SYSTEM FillingModule (* Module Filling, generated from its module specification *)
  (* Standard: 61499-2 *)
  APPLICATION Filling (* Module Filling on target pc (localhost, IO modbus; generated by modgen) *)
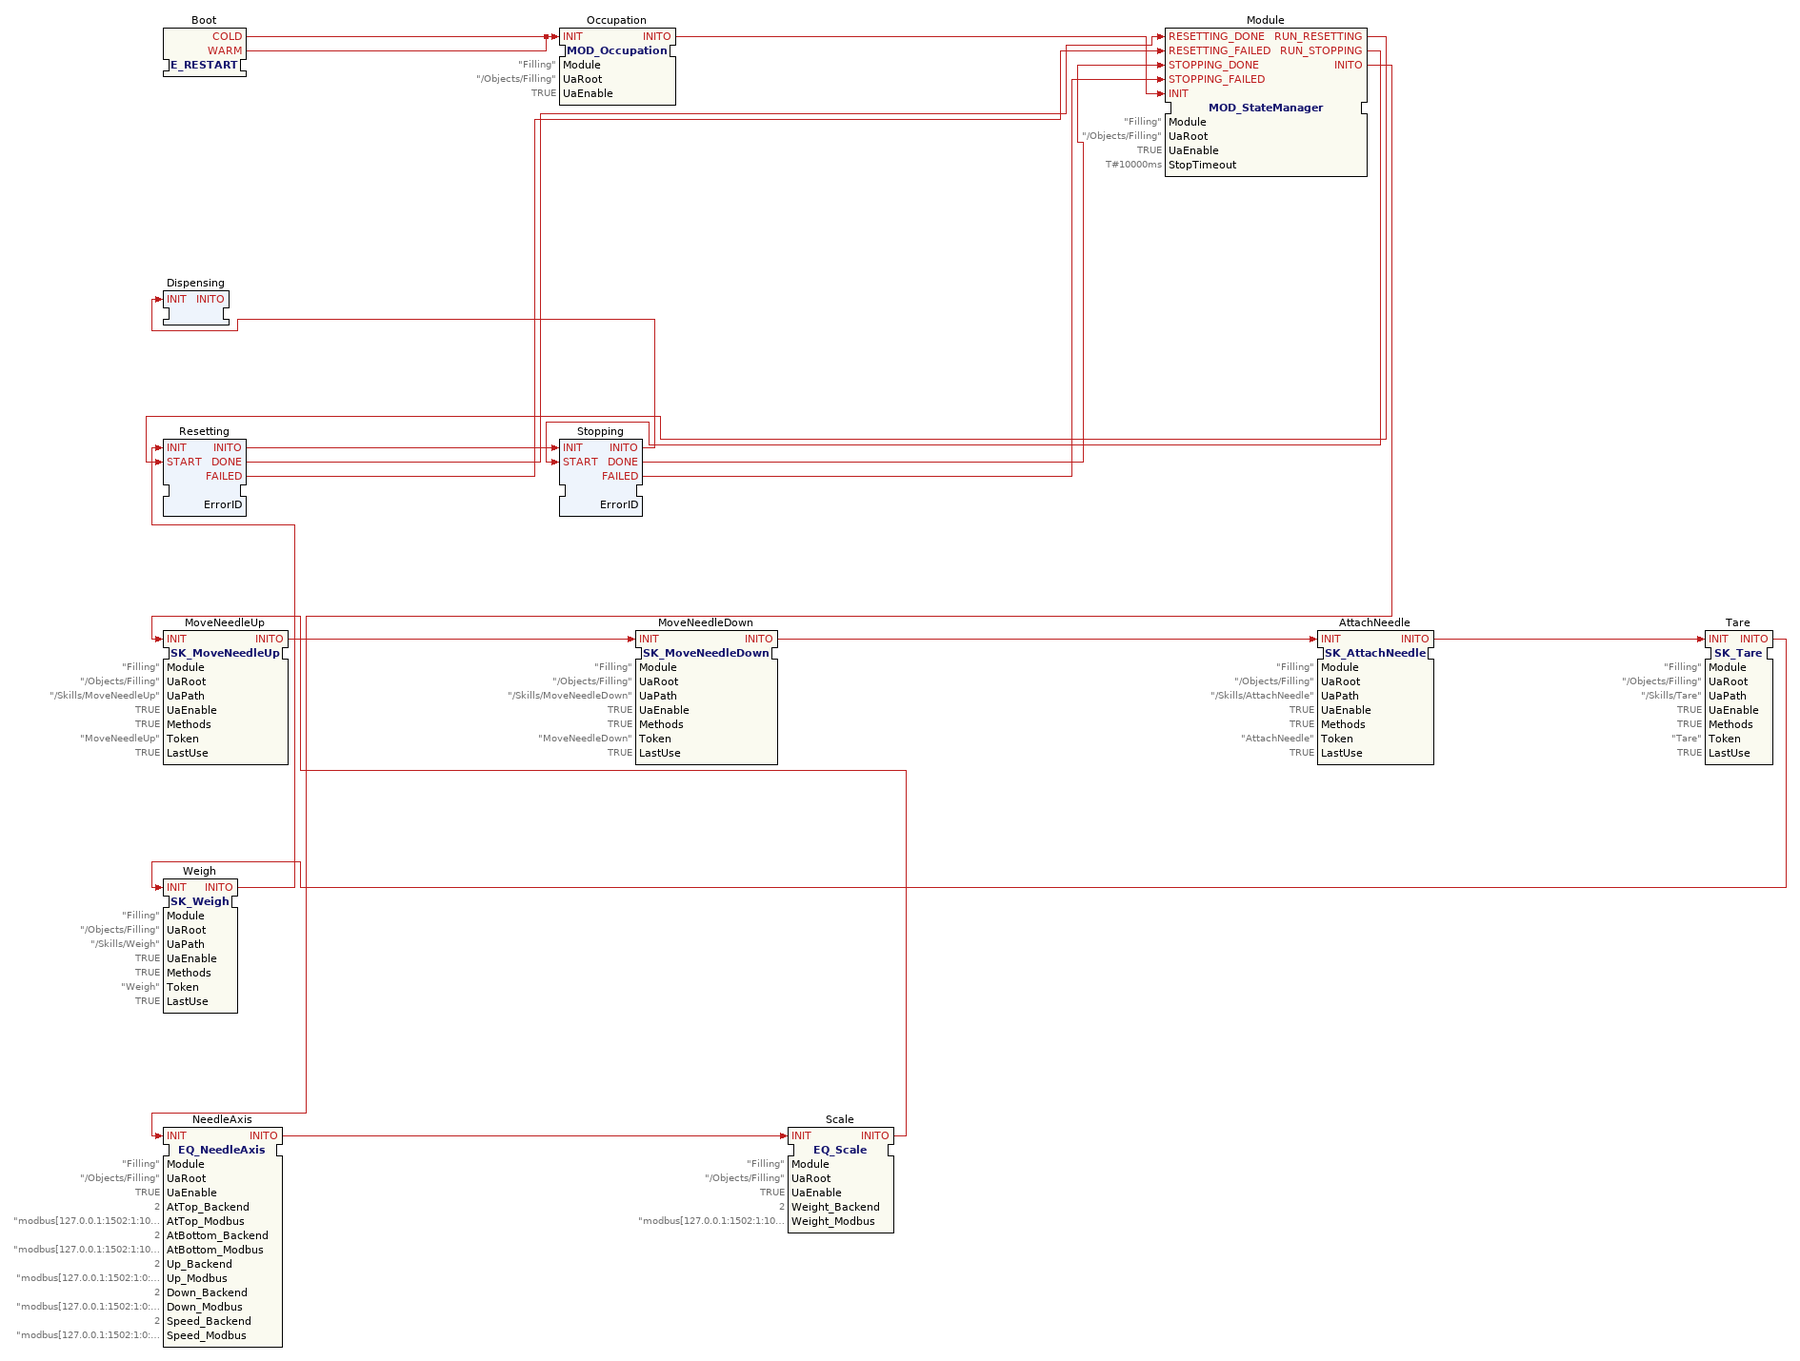
    (* Group ModuleLevel: Module level: occupation, PackML state manager, start-up and the target's IO lines *)
    (* Group ModuleLevelSkills: Module level skills: Control, Sequences (Execute, Stop) of skill primitives and Release; OPC UA /Skills/<name> *)
    (* Group Procedures: Procedures the module state manager runs while Resetting and Stopping *)
    (* Group SkillPrimitives: Skill primitives: one equipment command until a sensor or a time; OPC UA /Skills/<name> *)
    (* Group EquipmentIO: Equipment IO: the only owners of the IO points; skills send them output values over local channels *)
    FBS
      Boot : iec61499::events::E_RESTART; {SET_ATTRIBUTE(GroupName, ModuleLevel)}
      Occupation : modlib::MOD_Occupation(Module := "Filling", UaRoot := "/Objects/Filling", UaEnable := TRUE); {SET_ATTRIBUTE(GroupName, ModuleLevel)}
      Module : modlib::MOD_StateManager(Module := "Filling", UaRoot := "/Objects/Filling", UaEnable := TRUE, StopTimeout := T#10000ms); {SET_ATTRIBUTE(GroupName, ModuleLevel)}
      NeedleAxis : filling::EQ_NeedleAxis(Module := "Filling", UaRoot := "/Objects/Filling", UaEnable := TRUE, AtTop_Backend := 2, AtTop_Modbus := "modbus[127.0.0.1:1502:1:10:d0:]", AtBottom_Backend := 2, AtBottom_Modbus := "modbus[127.0.0.1:1502:1:10:d1:]", Up_Backend := 2, Up_Modbus := "modbus[127.0.0.1:1502:1:0::c0]", Down_Backend := 2, Down_Modbus := "modbus[127.0.0.1:1502:1:0::c1]", Speed_Backend := 2, Speed_Modbus := "modbus[127.0.0.1:1502:1:0::h0]"); {SET_ATTRIBUTE(GroupName, EquipmentIO)}
      Scale : filling::EQ_Scale(Module := "Filling", UaRoot := "/Objects/Filling", UaEnable := TRUE, Weight_Backend := 2, Weight_Modbus := "modbus[127.0.0.1:1502:1:10:i0:]"); {SET_ATTRIBUTE(GroupName, EquipmentIO)}
      MoveNeedleUp : filling::SK_MoveNeedleUp(Module := "Filling", UaRoot := "/Objects/Filling", UaPath := "/Skills/MoveNeedleUp", UaEnable := TRUE, Methods := TRUE, Token := "MoveNeedleUp", LastUse := TRUE); {SET_ATTRIBUTE(GroupName, SkillPrimitives)}
      MoveNeedleDown : filling::SK_MoveNeedleDown(Module := "Filling", UaRoot := "/Objects/Filling", UaPath := "/Skills/MoveNeedleDown", UaEnable := TRUE, Methods := TRUE, Token := "MoveNeedleDown", LastUse := TRUE); {SET_ATTRIBUTE(GroupName, SkillPrimitives)}
      AttachNeedle : filling::SK_AttachNeedle(Module := "Filling", UaRoot := "/Objects/Filling", UaPath := "/Skills/AttachNeedle", UaEnable := TRUE, Methods := TRUE, Token := "AttachNeedle", LastUse := TRUE); {SET_ATTRIBUTE(GroupName, SkillPrimitives)}
      Tare : filling::SK_Tare(Module := "Filling", UaRoot := "/Objects/Filling", UaPath := "/Skills/Tare", UaEnable := TRUE, Methods := TRUE, Token := "Tare", LastUse := TRUE); {SET_ATTRIBUTE(GroupName, SkillPrimitives)}
      Weigh : filling::SK_Weigh(Module := "Filling", UaRoot := "/Objects/Filling", UaPath := "/Skills/Weigh", UaEnable := TRUE, Methods := TRUE, Token := "Weigh", LastUse := TRUE); {SET_ATTRIBUTE(GroupName, SkillPrimitives)}
    END_FBS
    SUBAPPLICATION Resetting (* Procedure the module runs while Resetting *)
      {SET_ATTRIBUTE(GroupName, Procedures)}
      EVENT_INPUT
        INIT : EInit;
        START;
      END_EVENT
      EVENT_OUTPUT
        INITO : EInit;
        DONE;
        FAILED;
      END_EVENT
      VAR_OUTPUT
        ErrorID : UINT;
      END_VAR
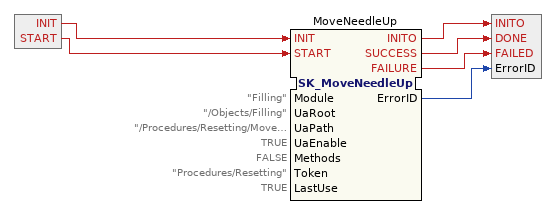
      FBS
        MoveNeedleUp : filling::SK_MoveNeedleUp(Module := "Filling", UaRoot := "/Objects/Filling", UaPath := "/Procedures/Resetting/MoveNeedleUp", UaEnable := TRUE, Methods := FALSE, Token := "Procedures/Resetting", LastUse := TRUE);
      END_FBS
      EVENT_CONNECTIONS
        INIT TO MoveNeedleUp.INIT;
        MoveNeedleUp.INITO TO INITO;
        START TO MoveNeedleUp.START;
        MoveNeedleUp.SUCCESS TO DONE;
        MoveNeedleUp.FAILURE TO FAILED;
      END_CONNECTIONS
      DATA_CONNECTIONS
        MoveNeedleUp.ErrorID TO ErrorID;
      END_CONNECTIONS
    END_SUBAPPLICATION
    SUBAPPLICATION Stopping (* Procedure the module runs while Stopping *)
      {SET_ATTRIBUTE(GroupName, Procedures)}
      EVENT_INPUT
        INIT : EInit;
        START;
      END_EVENT
      EVENT_OUTPUT
        INITO : EInit;
        DONE;
        FAILED;
      END_EVENT
      VAR_OUTPUT
        ErrorID : UINT;
      END_VAR
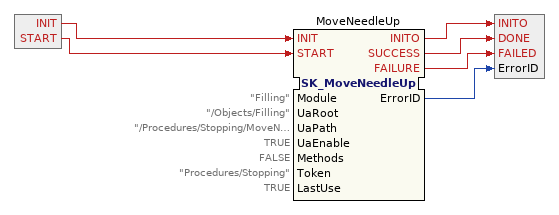
      FBS
        MoveNeedleUp : filling::SK_MoveNeedleUp(Module := "Filling", UaRoot := "/Objects/Filling", UaPath := "/Procedures/Stopping/MoveNeedleUp", UaEnable := TRUE, Methods := FALSE, Token := "Procedures/Stopping", LastUse := TRUE);
      END_FBS
      EVENT_CONNECTIONS
        INIT TO MoveNeedleUp.INIT;
        MoveNeedleUp.INITO TO INITO;
        START TO MoveNeedleUp.START;
        MoveNeedleUp.SUCCESS TO DONE;
        MoveNeedleUp.FAILURE TO FAILED;
      END_CONNECTIONS
      DATA_CONNECTIONS
        MoveNeedleUp.ErrorID TO ErrorID;
      END_CONNECTIONS
    END_SUBAPPLICATION
    SUBAPPLICATION Dispensing (* Module level skill Dispensing: Needle down, dispense the volume, needle up, weigh (runFillingCycle) *)
      {SET_ATTRIBUTE(GroupName, ModuleLevelSkills)}
      EVENT_INPUT
        INIT : EInit;
      END_EVENT
      EVENT_OUTPUT
        INITO : EInit;
      END_EVENT
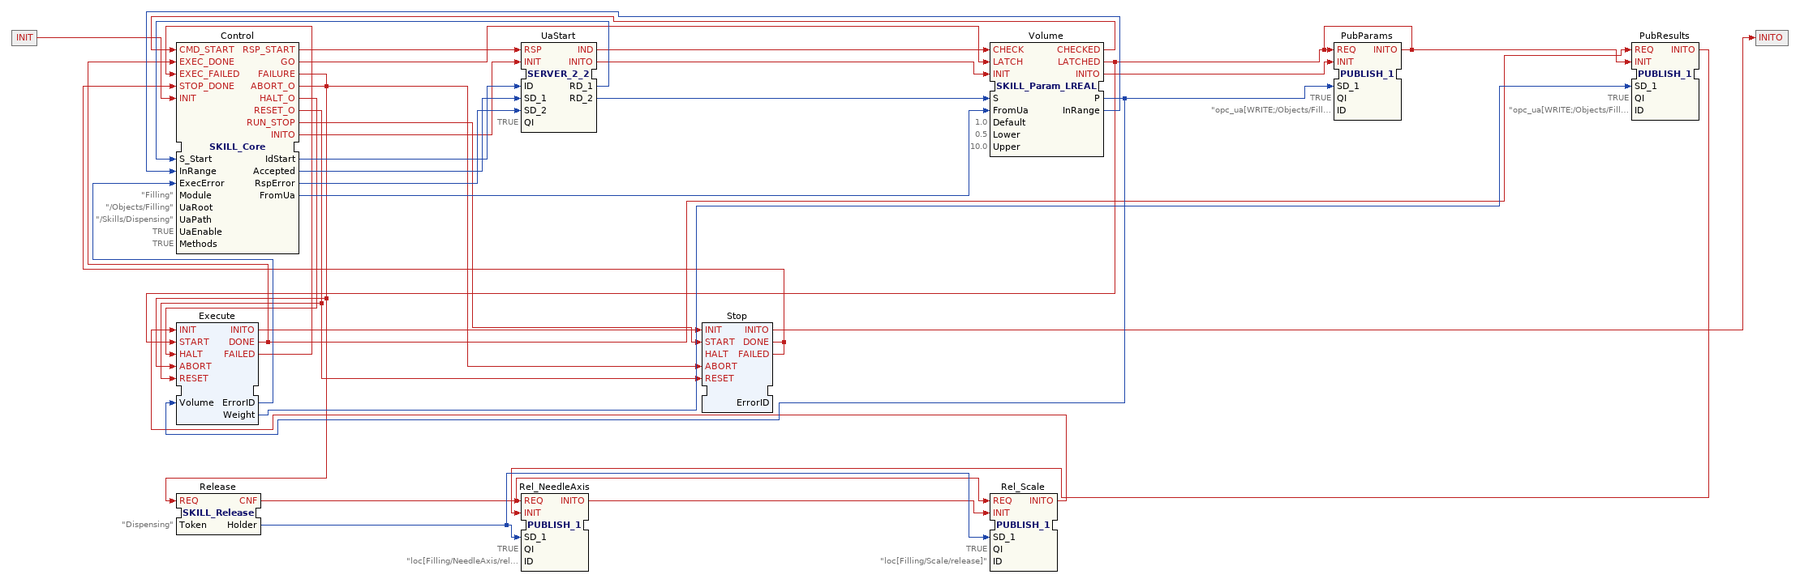
      (* Group SkillControl: State machine and OPC UA: Start(Session, parameters) with one block per parameter (range check, value for this run), Stop, Abort, Reset; State, parameters and results published *)
      (* Group Sequences: What the skill does: Execute, and Stop when it is interrupted; private skill primitives in order *)
      (* Group Releasing: After a failure or an abort: gives up the equipment the skill holds (all off, free again) *)
      FBS
        Control : modlib::SKILL_Core(Module := "Filling", UaRoot := "/Objects/Filling", UaPath := "/Skills/Dispensing", UaEnable := TRUE, Methods := TRUE); {SET_ATTRIBUTE(GroupName, SkillControl)}
        UaStart : iec61499::net::SERVER_2_2(QI := TRUE); {SET_ATTRIBUTE(GroupName, SkillControl)}
        Volume : modlib::SKILL_Param_LREAL(Default := 1.0, Lower := 0.5, Upper := 10.0); {SET_ATTRIBUTE(GroupName, SkillControl)}
        PubParams : iec61499::net::PUBLISH_1(QI := TRUE, ID := "opc_ua[WRITE;/Objects/Filling/Skills/Dispensing/Parameters/Volume]"); {SET_ATTRIBUTE(GroupName, SkillControl)}
        PubResults : iec61499::net::PUBLISH_1(QI := TRUE, ID := "opc_ua[WRITE;/Objects/Filling/Skills/Dispensing/Results/Weight]"); {SET_ATTRIBUTE(GroupName, SkillControl)}
        Release : modlib::SKILL_Release(Token := "Dispensing"); {SET_ATTRIBUTE(GroupName, Releasing)}
        Rel_NeedleAxis : iec61499::net::PUBLISH_1(QI := TRUE, ID := "loc[Filling/NeedleAxis/release]"); {SET_ATTRIBUTE(GroupName, Releasing)}
        Rel_Scale : iec61499::net::PUBLISH_1(QI := TRUE, ID := "loc[Filling/Scale/release]"); {SET_ATTRIBUTE(GroupName, Releasing)}
      END_FBS
      SUBAPPLICATION Execute (* Dispensing: execute sequence *)
        {SET_ATTRIBUTE(GroupName, Sequences)}
        EVENT_INPUT
          INIT : EInit;
          START;
          HALT;
          ABORT;
          RESET;
        END_EVENT
        EVENT_OUTPUT
          INITO : EInit;
          DONE;
          FAILED;
        END_EVENT
        VAR_INPUT
          Volume : LREAL;
        END_VAR
        VAR_OUTPUT
          ErrorID : UINT;
          Weight : LREAL;
        END_VAR
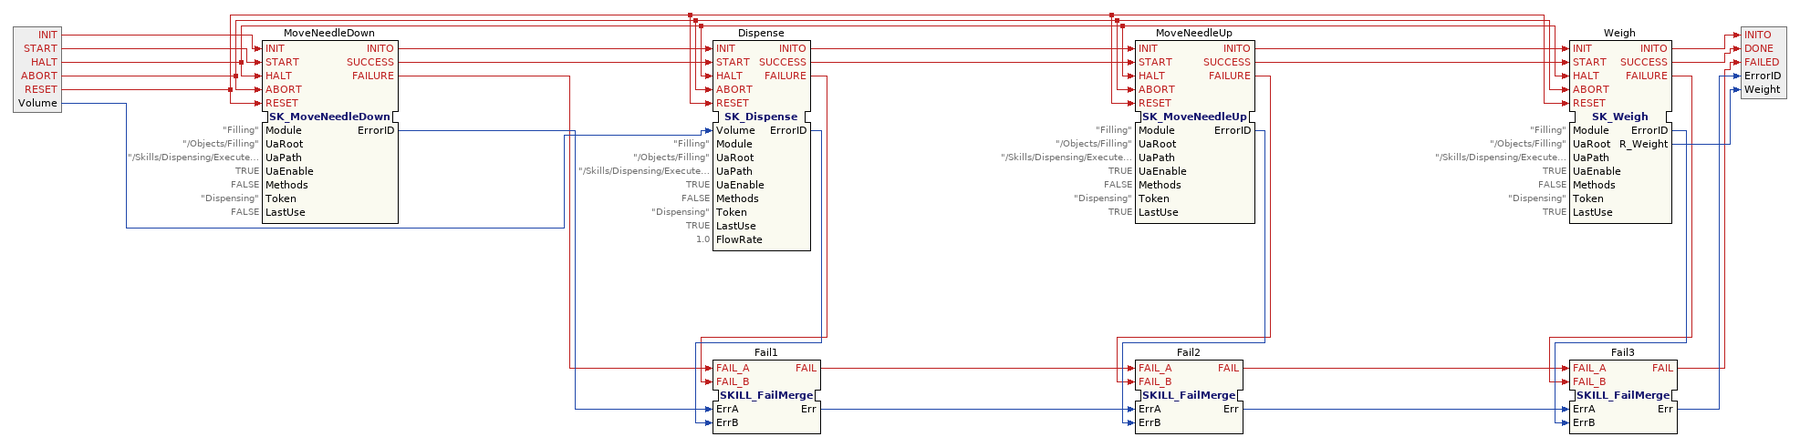
        FBS
          MoveNeedleDown : filling::SK_MoveNeedleDown(Module := "Filling", UaRoot := "/Objects/Filling", UaPath := "/Skills/Dispensing/Execute/MoveNeedleDown", UaEnable := TRUE, Methods := FALSE, Token := "Dispensing", LastUse := FALSE);
          Dispense : filling::SK_Dispense(Module := "Filling", UaRoot := "/Objects/Filling", UaPath := "/Skills/Dispensing/Execute/Dispense", UaEnable := TRUE, Methods := FALSE, Token := "Dispensing", LastUse := TRUE, FlowRate := 1.0);
          MoveNeedleUp : filling::SK_MoveNeedleUp(Module := "Filling", UaRoot := "/Objects/Filling", UaPath := "/Skills/Dispensing/Execute/MoveNeedleUp", UaEnable := TRUE, Methods := FALSE, Token := "Dispensing", LastUse := TRUE);
          Weigh : filling::SK_Weigh(Module := "Filling", UaRoot := "/Objects/Filling", UaPath := "/Skills/Dispensing/Execute/Weigh", UaEnable := TRUE, Methods := FALSE, Token := "Dispensing", LastUse := TRUE);
          Fail1 : modlib::SKILL_FailMerge;
          Fail2 : modlib::SKILL_FailMerge;
          Fail3 : modlib::SKILL_FailMerge;
        END_FBS
        EVENT_CONNECTIONS
          INIT TO MoveNeedleDown.INIT;
          Weigh.INITO TO INITO;
          START TO MoveNeedleDown.START;
          Weigh.SUCCESS TO DONE;
          MoveNeedleDown.INITO TO Dispense.INIT;
          MoveNeedleDown.SUCCESS TO Dispense.START;
          Dispense.INITO TO MoveNeedleUp.INIT;
          Dispense.SUCCESS TO MoveNeedleUp.START;
          MoveNeedleUp.INITO TO Weigh.INIT;
          MoveNeedleUp.SUCCESS TO Weigh.START;
          HALT TO MoveNeedleDown.HALT;
          HALT TO Dispense.HALT;
          HALT TO MoveNeedleUp.HALT;
          HALT TO Weigh.HALT;
          ABORT TO MoveNeedleDown.ABORT;
          ABORT TO Dispense.ABORT;
          ABORT TO MoveNeedleUp.ABORT;
          ABORT TO Weigh.ABORT;
          RESET TO MoveNeedleDown.RESET;
          RESET TO Dispense.RESET;
          RESET TO MoveNeedleUp.RESET;
          RESET TO Weigh.RESET;
          MoveNeedleDown.FAILURE TO Fail1.FAIL_A;
          Dispense.FAILURE TO Fail1.FAIL_B;
          Fail1.FAIL TO Fail2.FAIL_A;
          MoveNeedleUp.FAILURE TO Fail2.FAIL_B;
          Fail2.FAIL TO Fail3.FAIL_A;
          Weigh.FAILURE TO Fail3.FAIL_B;
          Fail3.FAIL TO FAILED;
        END_CONNECTIONS
        DATA_CONNECTIONS
          MoveNeedleDown.ErrorID TO Fail1.ErrA;
          Dispense.ErrorID TO Fail1.ErrB;
          Fail1.Err TO Fail2.ErrA;
          MoveNeedleUp.ErrorID TO Fail2.ErrB;
          Fail2.Err TO Fail3.ErrA;
          Weigh.ErrorID TO Fail3.ErrB;
          Fail3.Err TO ErrorID;
          Volume TO Dispense.Volume;
          Weigh.R_Weight TO Weight;
        END_CONNECTIONS
      END_SUBAPPLICATION
      SUBAPPLICATION Stop (* Dispensing: stop sequence *)
        {SET_ATTRIBUTE(GroupName, Sequences)}
        EVENT_INPUT
          INIT : EInit;
          START;
          HALT;
          ABORT;
          RESET;
        END_EVENT
        EVENT_OUTPUT
          INITO : EInit;
          DONE;
          FAILED;
        END_EVENT
        VAR_OUTPUT
          ErrorID : UINT;
        END_VAR
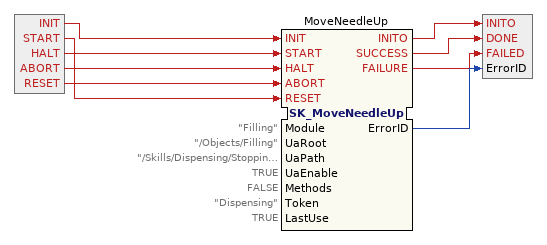
        FBS
          MoveNeedleUp : filling::SK_MoveNeedleUp(Module := "Filling", UaRoot := "/Objects/Filling", UaPath := "/Skills/Dispensing/Stopping/MoveNeedleUp", UaEnable := TRUE, Methods := FALSE, Token := "Dispensing", LastUse := TRUE);
        END_FBS
        EVENT_CONNECTIONS
          INIT TO MoveNeedleUp.INIT;
          MoveNeedleUp.INITO TO INITO;
          START TO MoveNeedleUp.START;
          MoveNeedleUp.SUCCESS TO DONE;
          HALT TO MoveNeedleUp.HALT;
          ABORT TO MoveNeedleUp.ABORT;
          RESET TO MoveNeedleUp.RESET;
          MoveNeedleUp.FAILURE TO FAILED;
        END_CONNECTIONS
        DATA_CONNECTIONS
          MoveNeedleUp.ErrorID TO ErrorID;
        END_CONNECTIONS
      END_SUBAPPLICATION
      EVENT_CONNECTIONS
        Control.RSP_START TO UaStart.RSP;
        UaStart.IND TO Volume.CHECK;
        Control.GO TO Volume.LATCH;
        Volume.CHECKED TO Control.CMD_START;
        Volume.LATCHED TO PubParams.REQ;
        PubParams.INITO TO PubParams.REQ;
        Execute.DONE TO PubResults.REQ;
        Control.FAILURE TO Release.REQ;
        Control.ABORT_O TO Release.REQ;
        Release.CNF TO Rel_NeedleAxis.REQ;
        Release.CNF TO Rel_Scale.REQ;
        Volume.LATCHED TO Execute.START;
        Control.HALT_O TO Execute.HALT;
        Control.ABORT_O TO Execute.ABORT;
        Control.RESET_O TO Execute.RESET;
        Execute.DONE TO Control.EXEC_DONE;
        Execute.FAILED TO Control.EXEC_FAILED;
        Control.RUN_STOP TO Stop.START;
        Control.ABORT_O TO Stop.ABORT;
        Control.RESET_O TO Stop.RESET;
        Stop.DONE TO Control.STOP_DONE;
        Stop.FAILED TO Control.STOP_DONE;
        INIT TO Control.INIT;
        Control.INITO TO UaStart.INIT;
        UaStart.INITO TO Volume.INIT;
        Volume.INITO TO PubParams.INIT;
        PubParams.INITO TO PubResults.INIT;
        PubResults.INITO TO Rel_NeedleAxis.INIT;
        Rel_NeedleAxis.INITO TO Rel_Scale.INIT;
        Rel_Scale.INITO TO Execute.INIT;
        Execute.INITO TO Stop.INIT;
        Stop.INITO TO INITO;
      END_CONNECTIONS
      DATA_CONNECTIONS
        Control.IdStart TO UaStart.ID;
        UaStart.RD_1 TO Control.S_Start;
        Control.Accepted TO UaStart.SD_1;
        Control.RspError TO UaStart.SD_2;
        UaStart.RD_2 TO Volume.S;
        Control.FromUa TO Volume.FromUa;
        Volume.P TO PubParams.SD_1;
        Volume.InRange TO Control.InRange;
        Execute.Weight TO PubResults.SD_1;
        Release.Holder TO Rel_NeedleAxis.SD_1;
        Release.Holder TO Rel_Scale.SD_1;
        Volume.P TO Execute.Volume;
        Execute.ErrorID TO Control.ExecError;
      END_CONNECTIONS
    END_SUBAPPLICATION
    EVENT_CONNECTIONS
      Boot.COLD TO Occupation.INIT;
      Boot.WARM TO Occupation.INIT;
      Module.RUN_RESETTING TO Resetting.START;
      Resetting.DONE TO Module.RESETTING_DONE;
      Resetting.FAILED TO Module.RESETTING_FAILED;
      Module.RUN_STOPPING TO Stopping.START;
      Stopping.DONE TO Module.STOPPING_DONE;
      Stopping.FAILED TO Module.STOPPING_FAILED;
      Occupation.INITO TO Module.INIT;
      Module.INITO TO NeedleAxis.INIT;
      NeedleAxis.INITO TO Scale.INIT;
      Scale.INITO TO MoveNeedleUp.INIT;
      MoveNeedleUp.INITO TO MoveNeedleDown.INIT;
      MoveNeedleDown.INITO TO AttachNeedle.INIT;
      AttachNeedle.INITO TO Tare.INIT;
      Tare.INITO TO Weigh.INIT;
      Weigh.INITO TO Resetting.INIT;
      Resetting.INITO TO Stopping.INIT;
      Stopping.INITO TO Dispensing.INIT;
    END_CONNECTIONS
  END_APPLICATION
  APPLICATION Filling_pi (* Module Filling on target pi (192.168.0.191, IO gpio; generated by modgen) *)
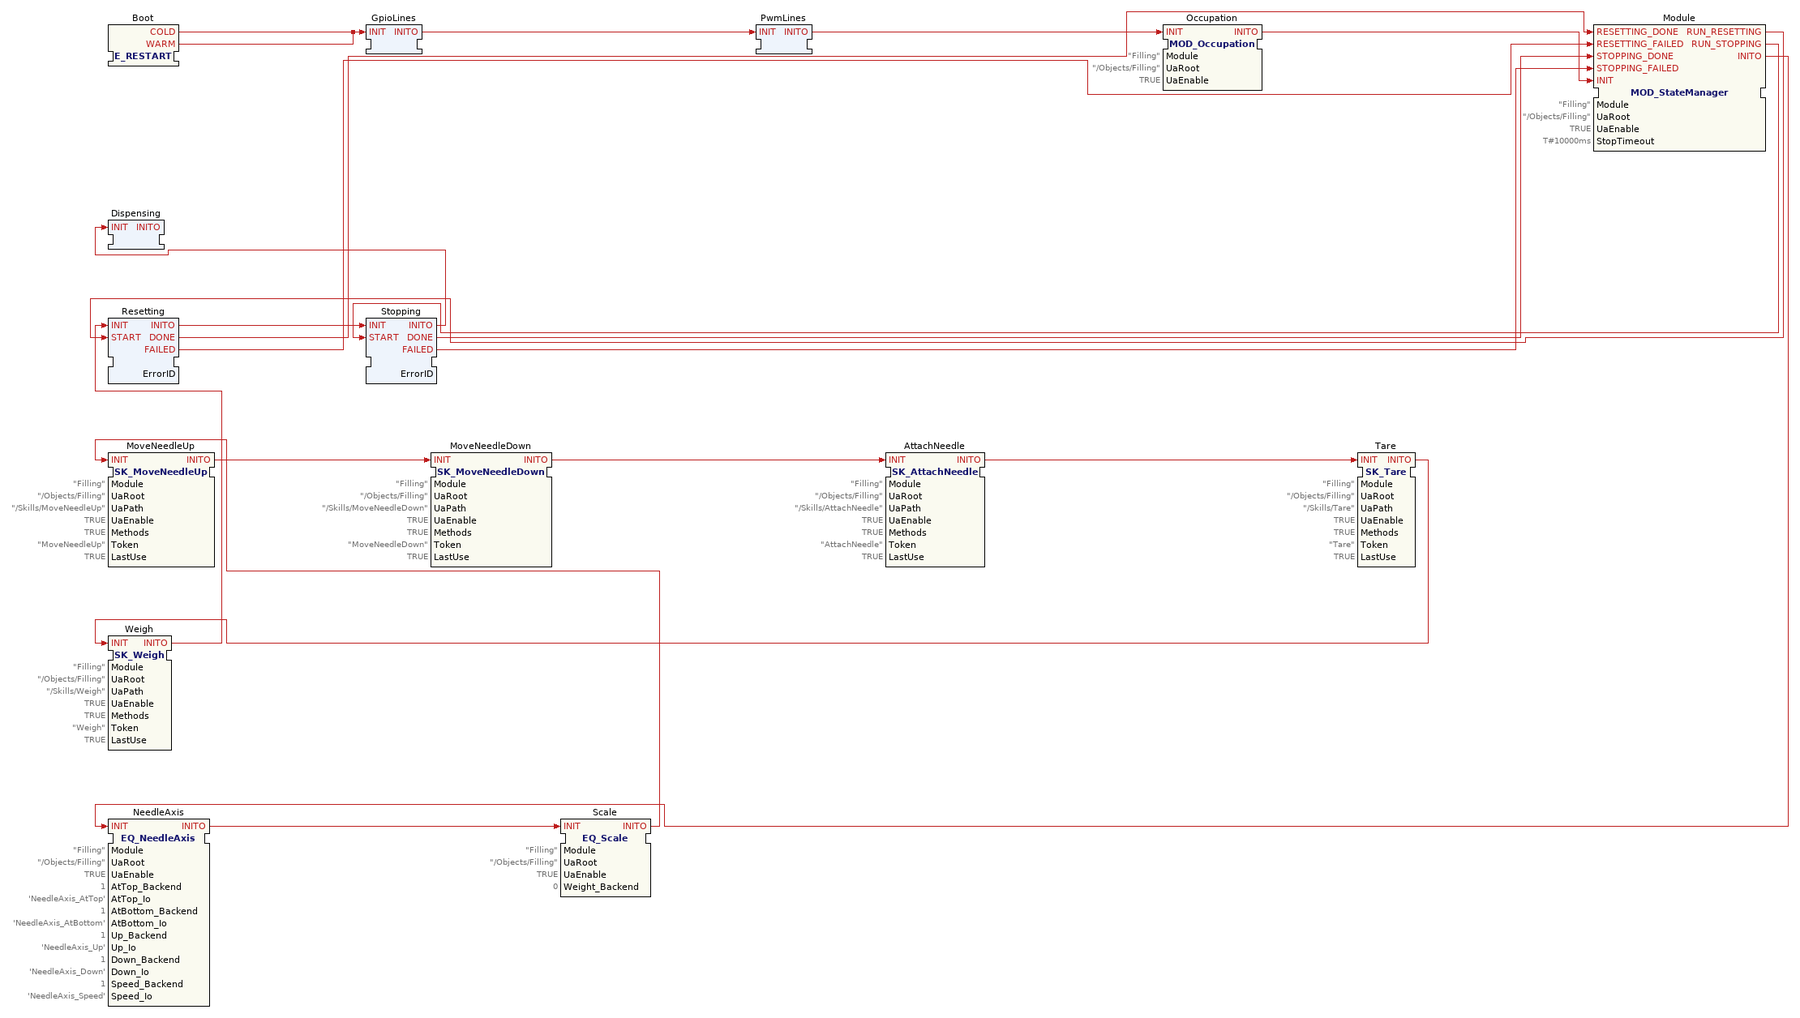
    (* Group ModuleLevel: Module level: occupation, PackML state manager, start-up and the target's IO lines *)
    (* Group ModuleLevelSkills: Module level skills: Control, Sequences (Execute, Stop) of skill primitives and Release; OPC UA /Skills/<name> *)
    (* Group Procedures: Procedures the module state manager runs while Resetting and Stopping *)
    (* Group SkillPrimitives: Skill primitives: one equipment command until a sensor or a time; OPC UA /Skills/<name> *)
    (* Group EquipmentIO: Equipment IO: the only owners of the IO points; skills send them output values over local channels *)
    FBS
      Boot : iec61499::events::E_RESTART; {SET_ATTRIBUTE(GroupName, ModuleLevel)}
      Occupation : modlib::MOD_Occupation(Module := "Filling", UaRoot := "/Objects/Filling", UaEnable := TRUE); {SET_ATTRIBUTE(GroupName, ModuleLevel)}
      Module : modlib::MOD_StateManager(Module := "Filling", UaRoot := "/Objects/Filling", UaEnable := TRUE, StopTimeout := T#10000ms); {SET_ATTRIBUTE(GroupName, ModuleLevel)}
      NeedleAxis : filling::EQ_NeedleAxis(Module := "Filling", UaRoot := "/Objects/Filling", UaEnable := TRUE, AtTop_Backend := 1, AtTop_Io := 'NeedleAxis_AtTop', AtBottom_Backend := 1, AtBottom_Io := 'NeedleAxis_AtBottom', Up_Backend := 1, Up_Io := 'NeedleAxis_Up', Down_Backend := 1, Down_Io := 'NeedleAxis_Down', Speed_Backend := 1, Speed_Io := 'NeedleAxis_Speed'); {SET_ATTRIBUTE(GroupName, EquipmentIO)}
      Scale : filling::EQ_Scale(Module := "Filling", UaRoot := "/Objects/Filling", UaEnable := TRUE, Weight_Backend := 0); {SET_ATTRIBUTE(GroupName, EquipmentIO)}
      MoveNeedleUp : filling::SK_MoveNeedleUp(Module := "Filling", UaRoot := "/Objects/Filling", UaPath := "/Skills/MoveNeedleUp", UaEnable := TRUE, Methods := TRUE, Token := "MoveNeedleUp", LastUse := TRUE); {SET_ATTRIBUTE(GroupName, SkillPrimitives)}
      MoveNeedleDown : filling::SK_MoveNeedleDown(Module := "Filling", UaRoot := "/Objects/Filling", UaPath := "/Skills/MoveNeedleDown", UaEnable := TRUE, Methods := TRUE, Token := "MoveNeedleDown", LastUse := TRUE); {SET_ATTRIBUTE(GroupName, SkillPrimitives)}
      AttachNeedle : filling::SK_AttachNeedle(Module := "Filling", UaRoot := "/Objects/Filling", UaPath := "/Skills/AttachNeedle", UaEnable := TRUE, Methods := TRUE, Token := "AttachNeedle", LastUse := TRUE); {SET_ATTRIBUTE(GroupName, SkillPrimitives)}
      Tare : filling::SK_Tare(Module := "Filling", UaRoot := "/Objects/Filling", UaPath := "/Skills/Tare", UaEnable := TRUE, Methods := TRUE, Token := "Tare", LastUse := TRUE); {SET_ATTRIBUTE(GroupName, SkillPrimitives)}
      Weigh : filling::SK_Weigh(Module := "Filling", UaRoot := "/Objects/Filling", UaPath := "/Skills/Weigh", UaEnable := TRUE, Methods := TRUE, Token := "Weigh", LastUse := TRUE); {SET_ATTRIBUTE(GroupName, SkillPrimitives)}
    END_FBS
    SUBAPPLICATION GpioLines (* GPIO lines of the equipment's IO points (Linux /dev/gpiochip) *)
      {SET_ATTRIBUTE(GroupName, ModuleLevel)}
      EVENT_INPUT
        INIT : EInit;
      END_EVENT
      EVENT_OUTPUT
        INITO : EInit;
      END_EVENT
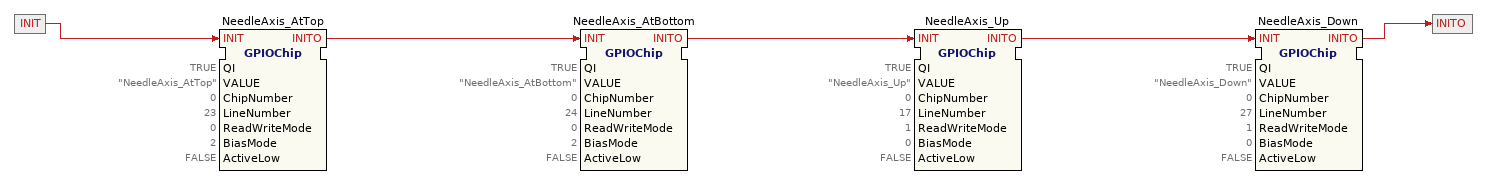
      FBS
        NeedleAxis_AtTop : eclipse4diac::io::gpiochip::GPIOChip(QI := TRUE, VALUE := "NeedleAxis_AtTop", ChipNumber := 0, LineNumber := 23, ReadWriteMode := 0, BiasMode := 2, ActiveLow := FALSE);
        NeedleAxis_AtBottom : eclipse4diac::io::gpiochip::GPIOChip(QI := TRUE, VALUE := "NeedleAxis_AtBottom", ChipNumber := 0, LineNumber := 24, ReadWriteMode := 0, BiasMode := 2, ActiveLow := FALSE);
        NeedleAxis_Up : eclipse4diac::io::gpiochip::GPIOChip(QI := TRUE, VALUE := "NeedleAxis_Up", ChipNumber := 0, LineNumber := 17, ReadWriteMode := 1, BiasMode := 0, ActiveLow := FALSE);
        NeedleAxis_Down : eclipse4diac::io::gpiochip::GPIOChip(QI := TRUE, VALUE := "NeedleAxis_Down", ChipNumber := 0, LineNumber := 27, ReadWriteMode := 1, BiasMode := 0, ActiveLow := FALSE);
      END_FBS
      EVENT_CONNECTIONS
        INIT TO NeedleAxis_AtTop.INIT;
        NeedleAxis_Down.INITO TO INITO;
        NeedleAxis_AtTop.INITO TO NeedleAxis_AtBottom.INIT;
        NeedleAxis_AtBottom.INITO TO NeedleAxis_Up.INIT;
        NeedleAxis_Up.INITO TO NeedleAxis_Down.INIT;
      END_CONNECTIONS
    END_SUBAPPLICATION
    SUBAPPLICATION PwmLines (* PWM channels of the equipment's analog outputs (Linux /sys/class/pwm) *)
      {SET_ATTRIBUTE(GroupName, ModuleLevel)}
      EVENT_INPUT
        INIT : EInit;
      END_EVENT
      EVENT_OUTPUT
        INITO : EInit;
      END_EVENT
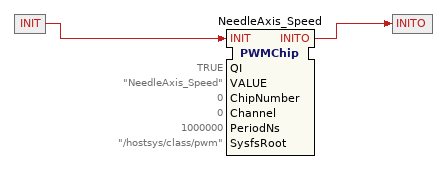
      FBS
        NeedleAxis_Speed : eclipse4diac::io::pwmsysfs::PWMChip(QI := TRUE, VALUE := "NeedleAxis_Speed", ChipNumber := 0, Channel := 0, PeriodNs := 1000000, SysfsRoot := "/hostsys/class/pwm");
      END_FBS
      EVENT_CONNECTIONS
        INIT TO NeedleAxis_Speed.INIT;
        NeedleAxis_Speed.INITO TO INITO;
      END_CONNECTIONS
    END_SUBAPPLICATION
    SUBAPPLICATION Resetting (* Procedure the module runs while Resetting *)
      {SET_ATTRIBUTE(GroupName, Procedures)}
      EVENT_INPUT
        INIT : EInit;
        START;
      END_EVENT
      EVENT_OUTPUT
        INITO : EInit;
        DONE;
        FAILED;
      END_EVENT
      VAR_OUTPUT
        ErrorID : UINT;
      END_VAR
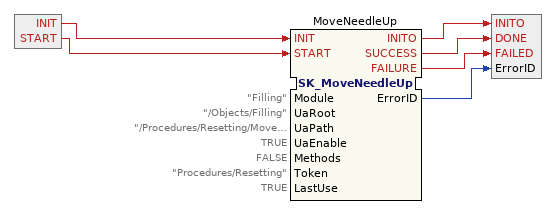
      FBS
        MoveNeedleUp : filling::SK_MoveNeedleUp(Module := "Filling", UaRoot := "/Objects/Filling", UaPath := "/Procedures/Resetting/MoveNeedleUp", UaEnable := TRUE, Methods := FALSE, Token := "Procedures/Resetting", LastUse := TRUE);
      END_FBS
      EVENT_CONNECTIONS
        INIT TO MoveNeedleUp.INIT;
        MoveNeedleUp.INITO TO INITO;
        START TO MoveNeedleUp.START;
        MoveNeedleUp.SUCCESS TO DONE;
        MoveNeedleUp.FAILURE TO FAILED;
      END_CONNECTIONS
      DATA_CONNECTIONS
        MoveNeedleUp.ErrorID TO ErrorID;
      END_CONNECTIONS
    END_SUBAPPLICATION
    SUBAPPLICATION Stopping (* Procedure the module runs while Stopping *)
      {SET_ATTRIBUTE(GroupName, Procedures)}
      EVENT_INPUT
        INIT : EInit;
        START;
      END_EVENT
      EVENT_OUTPUT
        INITO : EInit;
        DONE;
        FAILED;
      END_EVENT
      VAR_OUTPUT
        ErrorID : UINT;
      END_VAR
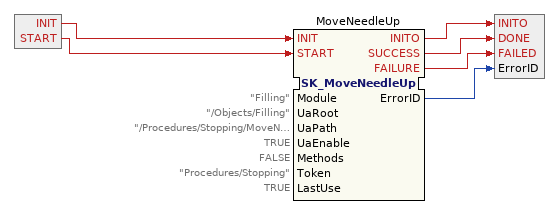
      FBS
        MoveNeedleUp : filling::SK_MoveNeedleUp(Module := "Filling", UaRoot := "/Objects/Filling", UaPath := "/Procedures/Stopping/MoveNeedleUp", UaEnable := TRUE, Methods := FALSE, Token := "Procedures/Stopping", LastUse := TRUE);
      END_FBS
      EVENT_CONNECTIONS
        INIT TO MoveNeedleUp.INIT;
        MoveNeedleUp.INITO TO INITO;
        START TO MoveNeedleUp.START;
        MoveNeedleUp.SUCCESS TO DONE;
        MoveNeedleUp.FAILURE TO FAILED;
      END_CONNECTIONS
      DATA_CONNECTIONS
        MoveNeedleUp.ErrorID TO ErrorID;
      END_CONNECTIONS
    END_SUBAPPLICATION
    SUBAPPLICATION Dispensing (* Module level skill Dispensing: Needle down, dispense the volume, needle up, weigh (runFillingCycle) *)
      {SET_ATTRIBUTE(GroupName, ModuleLevelSkills)}
      EVENT_INPUT
        INIT : EInit;
      END_EVENT
      EVENT_OUTPUT
        INITO : EInit;
      END_EVENT
      (* Group SkillControl: State machine and OPC UA: Start(Session, parameters) with one block per parameter (range check, value for this run), Stop, Abort, Reset; State, parameters and results published *)
      (* Group Sequences: What the skill does: Execute, and Stop when it is interrupted; private skill primitives in order *)
      (* Group Releasing: After a failure or an abort: gives up the equipment the skill holds (all off, free again) *)
      FBS
        Control : modlib::SKILL_Core(Module := "Filling", UaRoot := "/Objects/Filling", UaPath := "/Skills/Dispensing", UaEnable := TRUE, Methods := TRUE); {SET_ATTRIBUTE(GroupName, SkillControl)}
        UaStart : iec61499::net::SERVER_2_2(QI := TRUE); {SET_ATTRIBUTE(GroupName, SkillControl)}
        Volume : modlib::SKILL_Param_LREAL(Default := 1.0, Lower := 0.5, Upper := 10.0); {SET_ATTRIBUTE(GroupName, SkillControl)}
        PubParams : iec61499::net::PUBLISH_1(QI := TRUE, ID := "opc_ua[WRITE;/Objects/Filling/Skills/Dispensing/Parameters/Volume]"); {SET_ATTRIBUTE(GroupName, SkillControl)}
        PubResults : iec61499::net::PUBLISH_1(QI := TRUE, ID := "opc_ua[WRITE;/Objects/Filling/Skills/Dispensing/Results/Weight]"); {SET_ATTRIBUTE(GroupName, SkillControl)}
        Release : modlib::SKILL_Release(Token := "Dispensing"); {SET_ATTRIBUTE(GroupName, Releasing)}
        Rel_NeedleAxis : iec61499::net::PUBLISH_1(QI := TRUE, ID := "loc[Filling/NeedleAxis/release]"); {SET_ATTRIBUTE(GroupName, Releasing)}
        Rel_Scale : iec61499::net::PUBLISH_1(QI := TRUE, ID := "loc[Filling/Scale/release]"); {SET_ATTRIBUTE(GroupName, Releasing)}
      END_FBS
      SUBAPPLICATION Execute (* Dispensing: execute sequence *)
        {SET_ATTRIBUTE(GroupName, Sequences)}
        EVENT_INPUT
          INIT : EInit;
          START;
          HALT;
          ABORT;
          RESET;
        END_EVENT
        EVENT_OUTPUT
          INITO : EInit;
          DONE;
          FAILED;
        END_EVENT
        VAR_INPUT
          Volume : LREAL;
        END_VAR
        VAR_OUTPUT
          ErrorID : UINT;
          Weight : LREAL;
        END_VAR
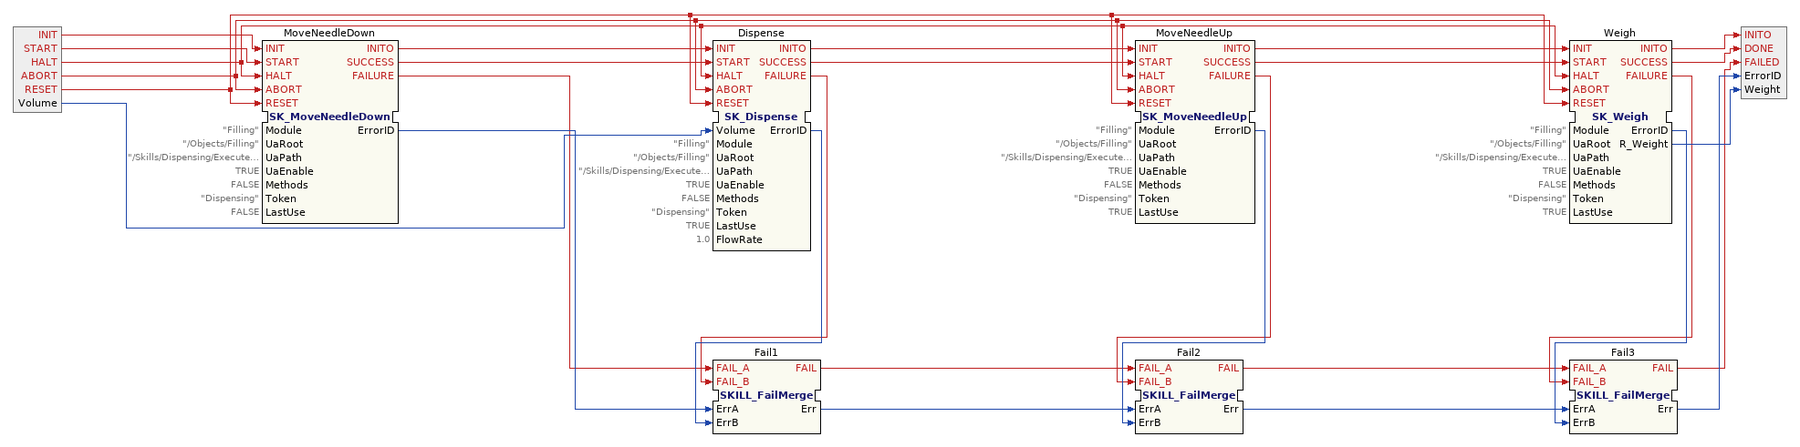
        FBS
          MoveNeedleDown : filling::SK_MoveNeedleDown(Module := "Filling", UaRoot := "/Objects/Filling", UaPath := "/Skills/Dispensing/Execute/MoveNeedleDown", UaEnable := TRUE, Methods := FALSE, Token := "Dispensing", LastUse := FALSE);
          Dispense : filling::SK_Dispense(Module := "Filling", UaRoot := "/Objects/Filling", UaPath := "/Skills/Dispensing/Execute/Dispense", UaEnable := TRUE, Methods := FALSE, Token := "Dispensing", LastUse := TRUE, FlowRate := 1.0);
          MoveNeedleUp : filling::SK_MoveNeedleUp(Module := "Filling", UaRoot := "/Objects/Filling", UaPath := "/Skills/Dispensing/Execute/MoveNeedleUp", UaEnable := TRUE, Methods := FALSE, Token := "Dispensing", LastUse := TRUE);
          Weigh : filling::SK_Weigh(Module := "Filling", UaRoot := "/Objects/Filling", UaPath := "/Skills/Dispensing/Execute/Weigh", UaEnable := TRUE, Methods := FALSE, Token := "Dispensing", LastUse := TRUE);
          Fail1 : modlib::SKILL_FailMerge;
          Fail2 : modlib::SKILL_FailMerge;
          Fail3 : modlib::SKILL_FailMerge;
        END_FBS
        EVENT_CONNECTIONS
          INIT TO MoveNeedleDown.INIT;
          Weigh.INITO TO INITO;
          START TO MoveNeedleDown.START;
          Weigh.SUCCESS TO DONE;
          MoveNeedleDown.INITO TO Dispense.INIT;
          MoveNeedleDown.SUCCESS TO Dispense.START;
          Dispense.INITO TO MoveNeedleUp.INIT;
          Dispense.SUCCESS TO MoveNeedleUp.START;
          MoveNeedleUp.INITO TO Weigh.INIT;
          MoveNeedleUp.SUCCESS TO Weigh.START;
          HALT TO MoveNeedleDown.HALT;
          HALT TO Dispense.HALT;
          HALT TO MoveNeedleUp.HALT;
          HALT TO Weigh.HALT;
          ABORT TO MoveNeedleDown.ABORT;
          ABORT TO Dispense.ABORT;
          ABORT TO MoveNeedleUp.ABORT;
          ABORT TO Weigh.ABORT;
          RESET TO MoveNeedleDown.RESET;
          RESET TO Dispense.RESET;
          RESET TO MoveNeedleUp.RESET;
          RESET TO Weigh.RESET;
          MoveNeedleDown.FAILURE TO Fail1.FAIL_A;
          Dispense.FAILURE TO Fail1.FAIL_B;
          Fail1.FAIL TO Fail2.FAIL_A;
          MoveNeedleUp.FAILURE TO Fail2.FAIL_B;
          Fail2.FAIL TO Fail3.FAIL_A;
          Weigh.FAILURE TO Fail3.FAIL_B;
          Fail3.FAIL TO FAILED;
        END_CONNECTIONS
        DATA_CONNECTIONS
          MoveNeedleDown.ErrorID TO Fail1.ErrA;
          Dispense.ErrorID TO Fail1.ErrB;
          Fail1.Err TO Fail2.ErrA;
          MoveNeedleUp.ErrorID TO Fail2.ErrB;
          Fail2.Err TO Fail3.ErrA;
          Weigh.ErrorID TO Fail3.ErrB;
          Fail3.Err TO ErrorID;
          Volume TO Dispense.Volume;
          Weigh.R_Weight TO Weight;
        END_CONNECTIONS
      END_SUBAPPLICATION
      SUBAPPLICATION Stop (* Dispensing: stop sequence *)
        {SET_ATTRIBUTE(GroupName, Sequences)}
        EVENT_INPUT
          INIT : EInit;
          START;
          HALT;
          ABORT;
          RESET;
        END_EVENT
        EVENT_OUTPUT
          INITO : EInit;
          DONE;
          FAILED;
        END_EVENT
        VAR_OUTPUT
          ErrorID : UINT;
        END_VAR
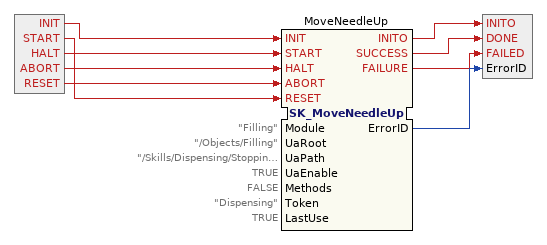
        FBS
          MoveNeedleUp : filling::SK_MoveNeedleUp(Module := "Filling", UaRoot := "/Objects/Filling", UaPath := "/Skills/Dispensing/Stopping/MoveNeedleUp", UaEnable := TRUE, Methods := FALSE, Token := "Dispensing", LastUse := TRUE);
        END_FBS
        EVENT_CONNECTIONS
          INIT TO MoveNeedleUp.INIT;
          MoveNeedleUp.INITO TO INITO;
          START TO MoveNeedleUp.START;
          MoveNeedleUp.SUCCESS TO DONE;
          HALT TO MoveNeedleUp.HALT;
          ABORT TO MoveNeedleUp.ABORT;
          RESET TO MoveNeedleUp.RESET;
          MoveNeedleUp.FAILURE TO FAILED;
        END_CONNECTIONS
        DATA_CONNECTIONS
          MoveNeedleUp.ErrorID TO ErrorID;
        END_CONNECTIONS
      END_SUBAPPLICATION
      EVENT_CONNECTIONS
        Control.RSP_START TO UaStart.RSP;
        UaStart.IND TO Volume.CHECK;
        Control.GO TO Volume.LATCH;
        Volume.CHECKED TO Control.CMD_START;
        Volume.LATCHED TO PubParams.REQ;
        PubParams.INITO TO PubParams.REQ;
        Execute.DONE TO PubResults.REQ;
        Control.FAILURE TO Release.REQ;
        Control.ABORT_O TO Release.REQ;
        Release.CNF TO Rel_NeedleAxis.REQ;
        Release.CNF TO Rel_Scale.REQ;
        Volume.LATCHED TO Execute.START;
        Control.HALT_O TO Execute.HALT;
        Control.ABORT_O TO Execute.ABORT;
        Control.RESET_O TO Execute.RESET;
        Execute.DONE TO Control.EXEC_DONE;
        Execute.FAILED TO Control.EXEC_FAILED;
        Control.RUN_STOP TO Stop.START;
        Control.ABORT_O TO Stop.ABORT;
        Control.RESET_O TO Stop.RESET;
        Stop.DONE TO Control.STOP_DONE;
        Stop.FAILED TO Control.STOP_DONE;
        INIT TO Control.INIT;
        Control.INITO TO UaStart.INIT;
        UaStart.INITO TO Volume.INIT;
        Volume.INITO TO PubParams.INIT;
        PubParams.INITO TO PubResults.INIT;
        PubResults.INITO TO Rel_NeedleAxis.INIT;
        Rel_NeedleAxis.INITO TO Rel_Scale.INIT;
        Rel_Scale.INITO TO Execute.INIT;
        Execute.INITO TO Stop.INIT;
        Stop.INITO TO INITO;
      END_CONNECTIONS
      DATA_CONNECTIONS
        Control.IdStart TO UaStart.ID;
        UaStart.RD_1 TO Control.S_Start;
        Control.Accepted TO UaStart.SD_1;
        Control.RspError TO UaStart.SD_2;
        UaStart.RD_2 TO Volume.S;
        Control.FromUa TO Volume.FromUa;
        Volume.P TO PubParams.SD_1;
        Volume.InRange TO Control.InRange;
        Execute.Weight TO PubResults.SD_1;
        Release.Holder TO Rel_NeedleAxis.SD_1;
        Release.Holder TO Rel_Scale.SD_1;
        Volume.P TO Execute.Volume;
        Execute.ErrorID TO Control.ExecError;
      END_CONNECTIONS
    END_SUBAPPLICATION
    EVENT_CONNECTIONS
      Boot.COLD TO GpioLines.INIT;
      Boot.WARM TO GpioLines.INIT;
      Module.RUN_RESETTING TO Resetting.START;
      Resetting.DONE TO Module.RESETTING_DONE;
      Resetting.FAILED TO Module.RESETTING_FAILED;
      Module.RUN_STOPPING TO Stopping.START;
      Stopping.DONE TO Module.STOPPING_DONE;
      Stopping.FAILED TO Module.STOPPING_FAILED;
      GpioLines.INITO TO PwmLines.INIT;
      PwmLines.INITO TO Occupation.INIT;
      Occupation.INITO TO Module.INIT;
      Module.INITO TO NeedleAxis.INIT;
      NeedleAxis.INITO TO Scale.INIT;
      Scale.INITO TO MoveNeedleUp.INIT;
      MoveNeedleUp.INITO TO MoveNeedleDown.INIT;
      MoveNeedleDown.INITO TO AttachNeedle.INIT;
      AttachNeedle.INITO TO Tare.INIT;
      Tare.INITO TO Weigh.INIT;
      Weigh.INITO TO Resetting.INIT;
      Resetting.INITO TO Stopping.INIT;
      Stopping.INITO TO Dispensing.INIT;
    END_CONNECTIONS
  END_APPLICATION
  DEVICE FORTE_PC : iec61499::system::FORTE_PC(MGR_ID := "localhost:61499" (* Device manager socket ID *))
    {SET_ATTRIBUTE(Profile, HOLOBLOC)}
    RESOURCE RES : iec61499::system::EMB_RES
    END_RESOURCE
  END_DEVICE
  DEVICE FORTE_PI : iec61499::system::FORTE_PC(MGR_ID := "192.168.0.191:61499" (* Device manager socket ID *))
    {SET_ATTRIBUTE(Profile, HOLOBLOC)}
    RESOURCE RES : iec61499::system::EMB_RES
    END_RESOURCE
  END_DEVICE
  MAPPINGS
    Filling.Boot ON FORTE_PC.RES;
    Filling.Occupation ON FORTE_PC.RES;
    Filling.Module ON FORTE_PC.RES;
    Filling.NeedleAxis ON FORTE_PC.RES;
    Filling.Scale ON FORTE_PC.RES;
    Filling.MoveNeedleUp ON FORTE_PC.RES;
    Filling.MoveNeedleDown ON FORTE_PC.RES;
    Filling.AttachNeedle ON FORTE_PC.RES;
    Filling.Tare ON FORTE_PC.RES;
    Filling.Weigh ON FORTE_PC.RES;
    Filling.Resetting ON FORTE_PC.RES;
    Filling.Stopping ON FORTE_PC.RES;
    Filling.Dispensing ON FORTE_PC.RES;
    Filling_pi.Boot ON FORTE_PI.RES;
    Filling_pi.Occupation ON FORTE_PI.RES;
    Filling_pi.Module ON FORTE_PI.RES;
    Filling_pi.GpioLines ON FORTE_PI.RES;
    Filling_pi.PwmLines ON FORTE_PI.RES;
    Filling_pi.NeedleAxis ON FORTE_PI.RES;
    Filling_pi.Scale ON FORTE_PI.RES;
    Filling_pi.MoveNeedleUp ON FORTE_PI.RES;
    Filling_pi.MoveNeedleDown ON FORTE_PI.RES;
    Filling_pi.AttachNeedle ON FORTE_PI.RES;
    Filling_pi.Tare ON FORTE_PI.RES;
    Filling_pi.Weigh ON FORTE_PI.RES;
    Filling_pi.Resetting ON FORTE_PI.RES;
    Filling_pi.Stopping ON FORTE_PI.RES;
    Filling_pi.Dispensing ON FORTE_PI.RES;
  END_MAPPINGS
END_SYSTEM
